// TIA Portal V16 export
// export: Created 2021-12-01T20:36:20.7617108Z, ExportSetting WithDefaults, DisplayName Totally Integrated Automation Portal, DisplayVersion V16 Update 4, DisplayName TIA Portal Version Control Interface, DisplayVersion V16 Update 2, DisplayName TIA Portal Openness, DisplayVersion V16 Update 4, DisplayName SINAMICS Startdrive Advanced, DisplayVersion V16 Update 5, DisplayName SINAMICS Startdrive G130, G150, S120, S150, SINAMICS MV, S210, DisplayVersion V16 Update 5, DisplayName SINAMICS Startdrive G110M, G120, G120C, G120D, G120P, G115D, DisplayVersion V16 Update 5, DisplayName STEP 7 Professional, DisplayVersion V16 Update 4, DisplayName STEP 7 Safety, DisplayVersion V16, DisplayName WinCC Advanced, DisplayVersion V16 Update 4
FUNCTION "ST00240_2_FC" : Void   // FC124, LAD
TITLE = ST00240_2
{ S7_Optimized_Access := 'TRUE' }
VERSION : 0.1
// stored: AutoNumber true, IsIECCheckEnabled false, SetENOAutomatically false, UDAEnableTagReadback false
   VAR_IN_OUT
      OPMODE : "OPMODE_OUT_UDT";
      HMI_EXTENSION : "HMI_EXTENSION_PANEL_UDT";
   END_VAR
   VAR_TEMP
      EmptyHS : "RT_HANDSHAKE_UDT";
   END_VAR
BEGIN

REGION Network 1: Alarm
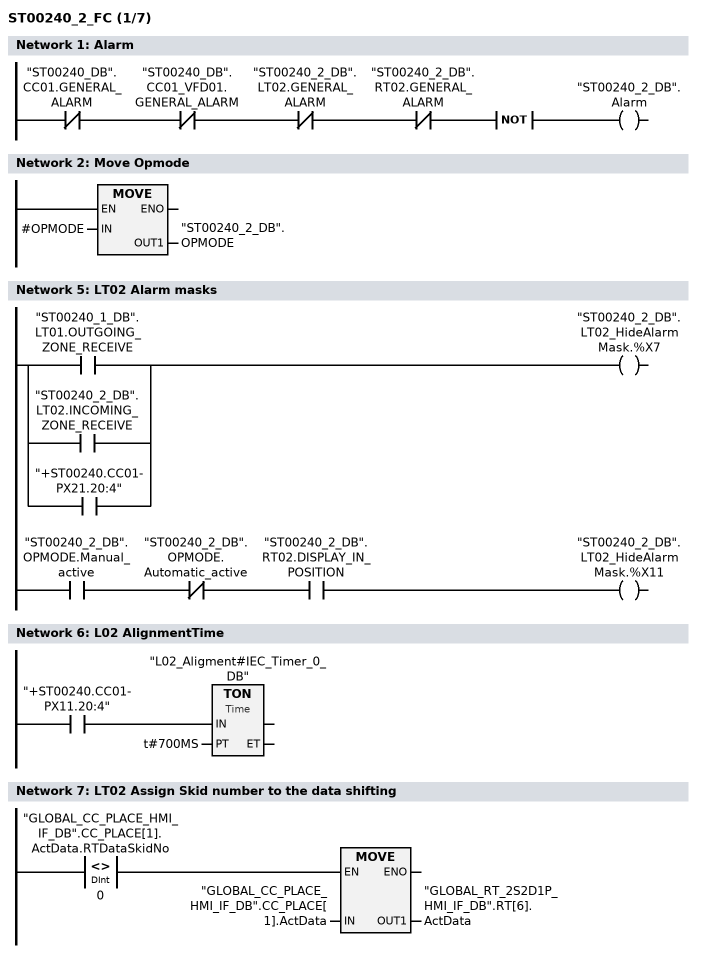
   RUNG wire#powerrail
      I_Contact( "ST00240_DB".CC01.GENERAL_ALARM )
      I_Contact( "ST00240_DB".CC01_VFD01.GENERAL_ALARM )
      I_Contact( "ST00240_2_DB".LT02.GENERAL_ALARM )
      I_Contact( "ST00240_2_DB".RT02.GENERAL_ALARM )
      Not()
      Coil( "ST00240_2_DB".Alarm )
   END_RUNG
   // the same network as SCL:
   "ST00240_2_DB".Alarm := NOT (NOT "ST00240_DB".CC01.GENERAL_ALARM AND NOT "ST00240_DB".CC01_VFD01.GENERAL_ALARM AND NOT "ST00240_2_DB".LT02.GENERAL_ALARM AND NOT "ST00240_2_DB".RT02.GENERAL_ALARM);
END_REGION

REGION Network 2: Move Opmode
   RUNG wire#powerrail
      Move(in := #OPMODE, out1 => "ST00240_2_DB".OPMODE)
   END_RUNG
   // the same network as SCL:
   "ST00240_2_DB".OPMODE := #OPMODE;
END_REGION

REGION Network 3: *******************LT02 Control*******************
END_REGION

REGION Network 4 (SCL): LT02 Parameters
   "ST00240_2_DB".LT02.PARA_SET.Para.HasMidPosition := true;
   "ST00240_2_DB".LT02.PARA_SET.Para.HasRT := TRUE;
   "ST00240_2_DB".LT02.PARA_SET.Para.PosCCStopForward := true;
   "ST00240_2_DB".LT02.PARA_SET.Para.PosCCStopReverse := false;
   "ST00240_2_DB".LT02.PARA_SET.Para.PosRaiseForward_1 := true;
   "ST00240_2_DB".LT02.PARA_SET.Para.PosRaiseForward_2 := true;
   "ST00240_2_DB".LT02.PARA_SET.Para.PosRaiseReverse_1 := true;
   "ST00240_2_DB".LT02.PARA_SET.Para.PosRaiseReverse_2 := false;
   "ST00240_2_DB".LT02.PARA_SET.Para.PosSlowForward := true;
   "ST00240_2_DB".LT02.PARA_SET.Para.PosSlowReverse := false;
   "ST00240_2_DB".LT02.PARA_SET.Set.RuntimeLower := t#10s;
   "ST00240_2_DB".LT02.PARA_SET.Set.RuntimeLift := t#11s;
   "ST00240_2_DB".LT02.PARA_SET.Set.AlignmentTime := t#0ms;
END_REGION

REGION Network 5: LT02 Alarm masks
   RUNG wire#powerrail
      Contact( "ST00240_1_DB".LT01.OUTGOING_ZONE_RECEIVE )
      wire#w1
      Coil( "ST00240_2_DB".LT02_HideAlarmMask.%X7 )
   END_RUNG
   RUNG wire#powerrail
      Contact( "ST00240_2_DB".LT02.INCOMING_ZONE_RECEIVE )
   END_RUNG wire#w1
   RUNG wire#powerrail
      Contact( "+ST00240.CC01-PX21.20:4" )
   END_RUNG wire#w1
   RUNG wire#powerrail
      Contact( "ST00240_2_DB".OPMODE.Manual_active )
      I_Contact( "ST00240_2_DB".OPMODE.Automatic_active )
      Contact( "ST00240_2_DB".RT02.DISPLAY_IN_POSITION )
      Coil( "ST00240_2_DB".LT02_HideAlarmMask.%X11 )
   END_RUNG
   // the same network as SCL:
   "ST00240_2_DB".LT02_HideAlarmMask.%X7 := "ST00240_1_DB".LT01.OUTGOING_ZONE_RECEIVE OR "ST00240_2_DB".LT02.INCOMING_ZONE_RECEIVE OR "+ST00240.CC01-PX21.20:4";
   "ST00240_2_DB".LT02_HideAlarmMask.%X11 := "ST00240_2_DB".OPMODE.Manual_active AND NOT "ST00240_2_DB".OPMODE.Automatic_active AND "ST00240_2_DB".RT02.DISPLAY_IN_POSITION;
END_REGION

REGION Network 6: L02 AlignmentTime
   RUNG wire#powerrail
      Contact( "+ST00240.CC01-PX11.20:4" )
      { S7_Templates := "time_type := Time" } "L02_Aligment#IEC_Timer_0_DB".TON(pt := t#700MS, et =>)
   END_RUNG
   // the same network as SCL:
   "L02_Aligment#IEC_Timer_0_DB".TON(IN := "+ST00240.CC01-PX11.20:4", PT := t#700MS);
END_REGION

REGION Network 7: LT02 Assign Skid number to the data shifting
   RUNG wire#powerrail
      { S7_Templates := "SrcType := DInt" } NE_Contact(in1 := "GLOBAL_CC_PLACE_HMI_IF_DB".CC_PLACE[1].ActData.RTDataSkidNo, in2 := 0)
      Move(in := "GLOBAL_CC_PLACE_HMI_IF_DB".CC_PLACE[1].ActData, out1 => "GLOBAL_RT_2S2D1P_HMI_IF_DB".RT[6].ActData)
   END_RUNG
   // the same network as SCL:
   IF "GLOBAL_CC_PLACE_HMI_IF_DB".CC_PLACE[1].ActData.RTDataSkidNo <> 0 THEN
       "GLOBAL_RT_2S2D1P_HMI_IF_DB".RT[6].ActData := "GLOBAL_CC_PLACE_HMI_IF_DB".CC_PLACE[1].ActData;
   END_IF;
END_REGION

REGION Network 8: LT02 CC Place FB
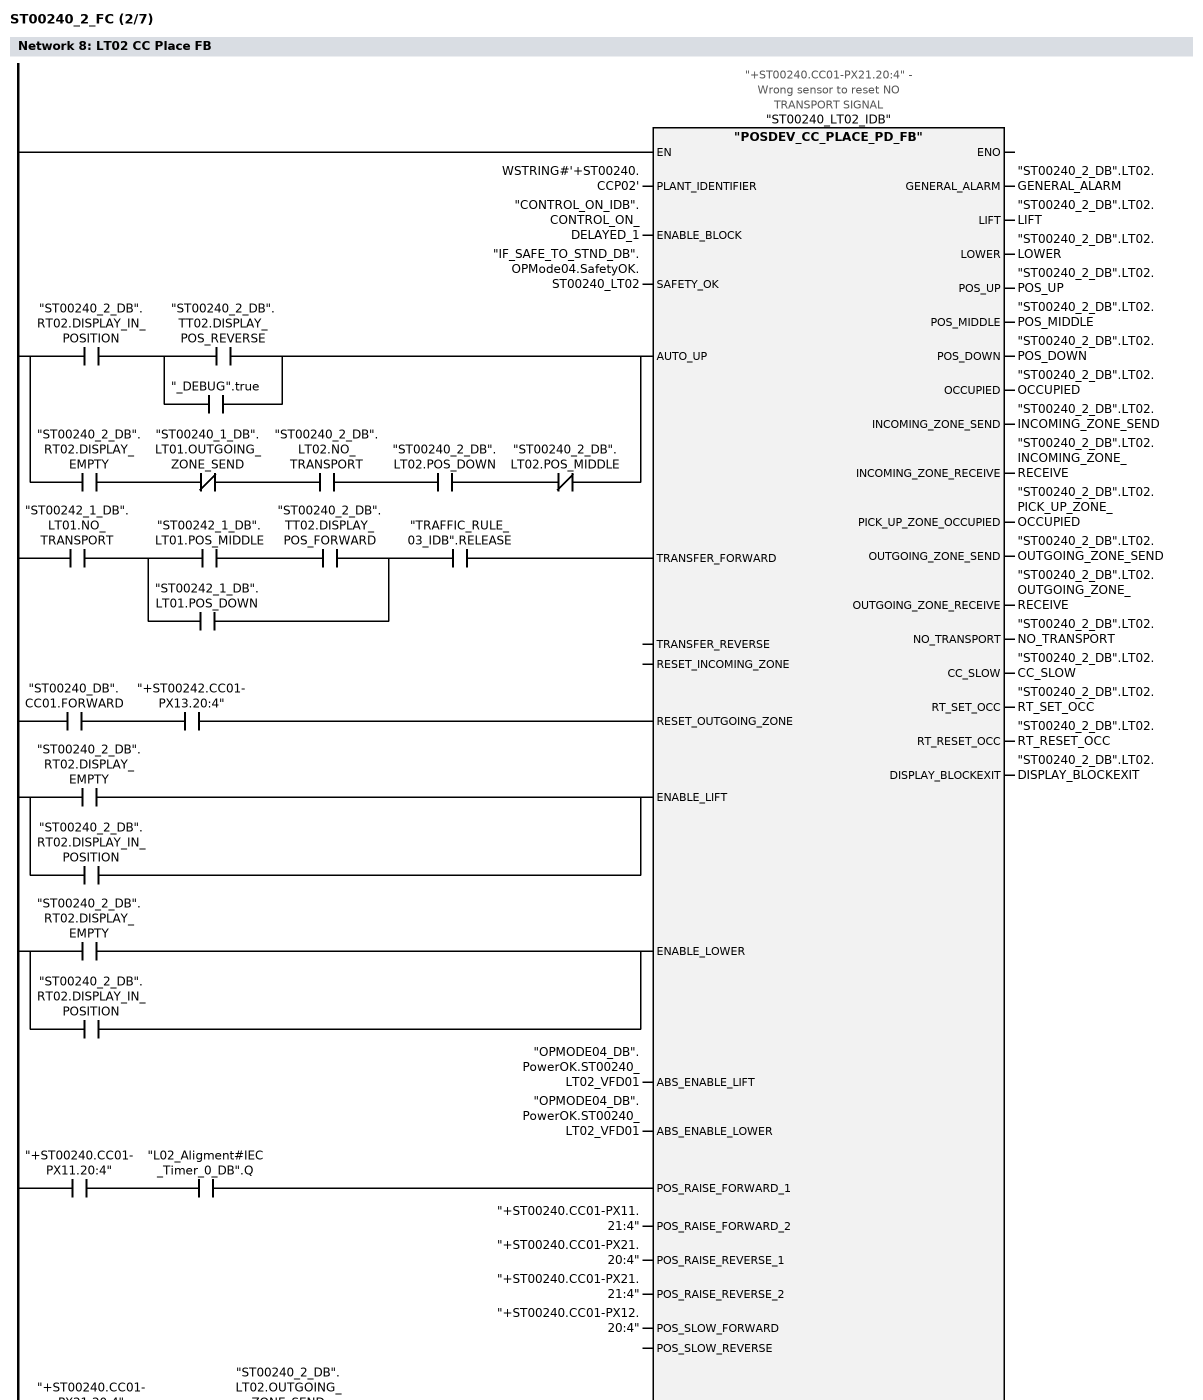
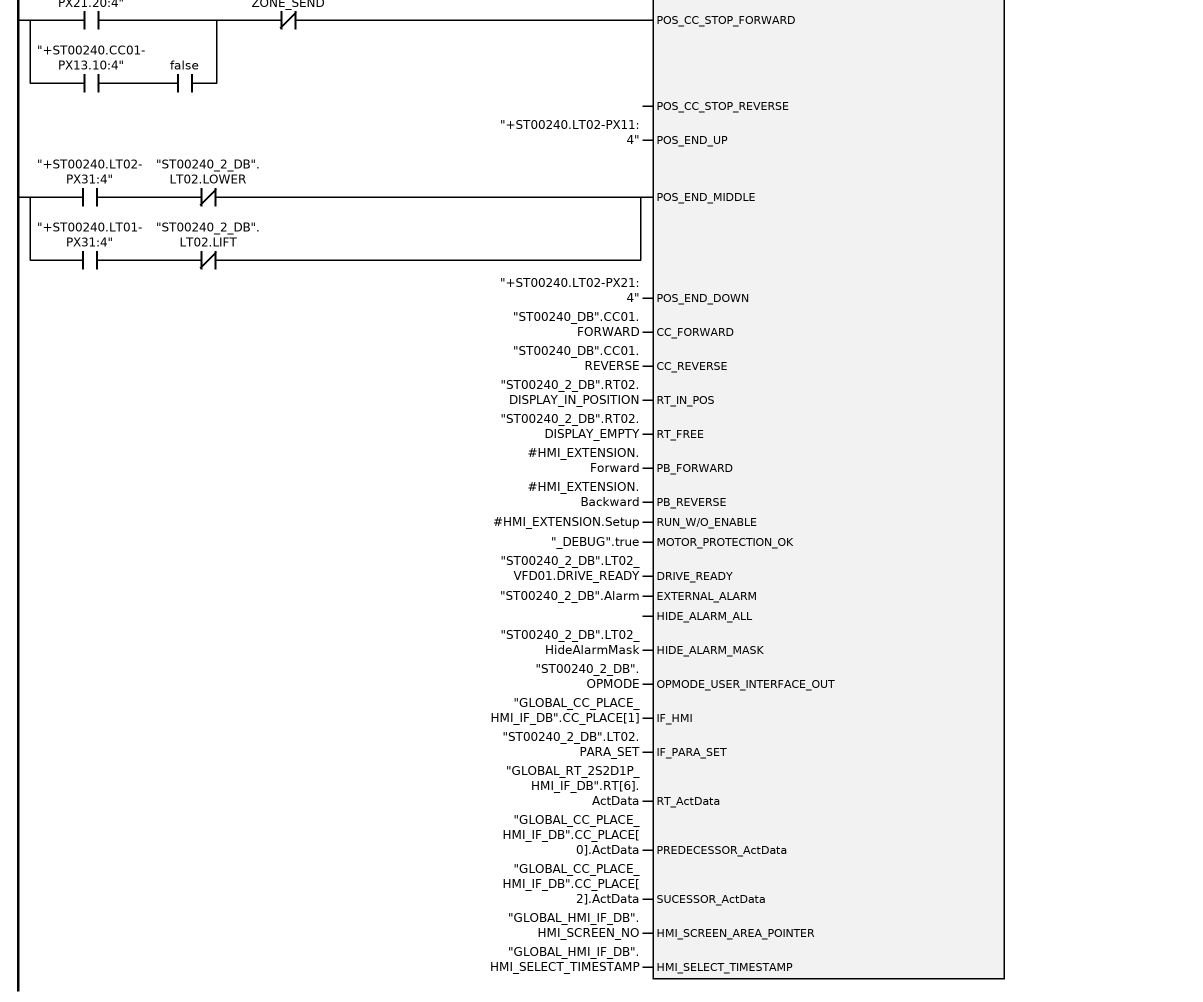
   RUNG wire#powerrail
      "ST00240_LT02_IDB"(AUTO_UP := wire#w2, TRANSFER_FORWARD := wire#w5, RESET_OUTGOING_ZONE := wire#w6, ENABLE_LIFT := wire#w7, ENABLE_LOWER := wire#w8, POS_RAISE_FORWARD_1 := wire#w9, POS_CC_STOP_FORWARD := wire#w11, POS_END_MIDDLE := wire#w12, PLANT_IDENTIFIER := WSTRING#'+ST00240.CCP02', ENABLE_BLOCK := "CONTROL_ON_IDB".CONTROL_ON_DELAYED_1, SAFETY_OK := "IF_SAFE_TO_STND_DB".OPMode04.SafetyOK.ST00240_LT02, TRANSFER_REVERSE :=, RESET_INCOMING_ZONE :=, ABS_ENABLE_LIFT := "OPMODE04_DB".PowerOK.ST00240_LT02_VFD01, ABS_ENABLE_LOWER := "OPMODE04_DB".PowerOK.ST00240_LT02_VFD01, POS_RAISE_FORWARD_2 := "+ST00240.CC01-PX11.21:4", POS_RAISE_REVERSE_1 := "+ST00240.CC01-PX21.20:4", POS_RAISE_REVERSE_2 := "+ST00240.CC01-PX21.21:4", POS_SLOW_FORWARD := "+ST00240.CC01-PX12.20:4", POS_SLOW_REVERSE :=, POS_CC_STOP_REVERSE :=, POS_END_UP := "+ST00240.LT02-PX11:4", POS_END_DOWN := "+ST00240.LT02-PX21:4", CC_FORWARD := "ST00240_DB".CC01.FORWARD, CC_REVERSE := "ST00240_DB".CC01.REVERSE, RT_IN_POS := "ST00240_2_DB".RT02.DISPLAY_IN_POSITION, RT_FREE := "ST00240_2_DB".RT02.DISPLAY_EMPTY, PB_FORWARD := #HMI_EXTENSION.Forward, PB_REVERSE := #HMI_EXTENSION.Backward, "RUN_W/O_ENABLE" := #HMI_EXTENSION.Setup, MOTOR_PROTECTION_OK := "_DEBUG".true, DRIVE_READY := "ST00240_2_DB".LT02_VFD01.DRIVE_READY, EXTERNAL_ALARM := "ST00240_2_DB".Alarm, HIDE_ALARM_ALL :=, HIDE_ALARM_MASK := "ST00240_2_DB".LT02_HideAlarmMask, OPMODE_USER_INTERFACE_OUT := "ST00240_2_DB".OPMODE, IF_HMI := "GLOBAL_CC_PLACE_HMI_IF_DB".CC_PLACE[1], IF_PARA_SET := "ST00240_2_DB".LT02.PARA_SET, RT_ActData := "GLOBAL_RT_2S2D1P_HMI_IF_DB".RT[6].ActData, PREDECESSOR_ActData := "GLOBAL_CC_PLACE_HMI_IF_DB".CC_PLACE[0].ActData, SUCESSOR_ActData := "GLOBAL_CC_PLACE_HMI_IF_DB".CC_PLACE[2].ActData, HMI_SCREEN_AREA_POINTER := "GLOBAL_HMI_IF_DB".HMI_SCREEN_NO, HMI_SELECT_TIMESTAMP := "GLOBAL_HMI_IF_DB".HMI_SELECT_TIMESTAMP, GENERAL_ALARM => "ST00240_2_DB".LT02.GENERAL_ALARM, LIFT => "ST00240_2_DB".LT02.LIFT, LOWER => "ST00240_2_DB".LT02.LOWER, POS_UP => "ST00240_2_DB".LT02.POS_UP, POS_MIDDLE => "ST00240_2_DB".LT02.POS_MIDDLE, POS_DOWN => "ST00240_2_DB".LT02.POS_DOWN, OCCUPIED => "ST00240_2_DB".LT02.OCCUPIED, INCOMING_ZONE_SEND => "ST00240_2_DB".LT02.INCOMING_ZONE_SEND, INCOMING_ZONE_RECEIVE => "ST00240_2_DB".LT02.INCOMING_ZONE_RECEIVE, PICK_UP_ZONE_OCCUPIED => "ST00240_2_DB".LT02.PICK_UP_ZONE_OCCUPIED, OUTGOING_ZONE_SEND => "ST00240_2_DB".LT02.OUTGOING_ZONE_SEND, OUTGOING_ZONE_RECEIVE => "ST00240_2_DB".LT02.OUTGOING_ZONE_RECEIVE, NO_TRANSPORT => "ST00240_2_DB".LT02.NO_TRANSPORT, CC_SLOW => "ST00240_2_DB".LT02.CC_SLOW, RT_SET_OCC => "ST00240_2_DB".LT02.RT_SET_OCC, RT_RESET_OCC => "ST00240_2_DB".LT02.RT_RESET_OCC, DISPLAY_BLOCKEXIT => "ST00240_2_DB".LT02.DISPLAY_BLOCKEXIT)   // "+ST00240.CC01-PX21.20:4" - Wrong sensor to reset NO TRANSPORT SIGNAL
   END_RUNG
   RUNG wire#powerrail
      Contact( "ST00240_2_DB".RT02.DISPLAY_IN_POSITION )
      wire#w1
      Contact( "ST00240_2_DB".TT02.DISPLAY_POS_REVERSE )
   END_RUNG wire#w2
   RUNG wire#w1
      Contact( "_DEBUG".true )
   END_RUNG wire#w2
   RUNG wire#powerrail
      Contact( "ST00240_2_DB".RT02.DISPLAY_EMPTY )
      I_Contact( "ST00240_1_DB".LT01.OUTGOING_ZONE_SEND )
      Contact( "ST00240_2_DB".LT02.NO_TRANSPORT )
      Contact( "ST00240_2_DB".LT02.POS_DOWN )
      I_Contact( "ST00240_2_DB".LT02.POS_MIDDLE )
   END_RUNG wire#w2
   RUNG wire#powerrail
      Contact( "ST00242_1_DB".LT01.NO_TRANSPORT )
      wire#w3
      Contact( "ST00242_1_DB".LT01.POS_MIDDLE )
      Contact( "ST00240_2_DB".TT02.DISPLAY_POS_FORWARD )
      wire#w4
      Contact( "TRAFFIC_RULE_03_IDB".RELEASE )
   END_RUNG wire#w5
   RUNG wire#w3
      Contact( "ST00242_1_DB".LT01.POS_DOWN )
   END_RUNG wire#w4
   RUNG wire#powerrail
      Contact( "ST00240_DB".CC01.FORWARD )
      Contact( "+ST00242.CC01-PX13.20:4" )
   END_RUNG wire#w6
   RUNG wire#powerrail
      Contact( "ST00240_2_DB".RT02.DISPLAY_EMPTY )
   END_RUNG wire#w7
   RUNG wire#powerrail
      Contact( "ST00240_2_DB".RT02.DISPLAY_IN_POSITION )
   END_RUNG wire#w7
   RUNG wire#powerrail
      Contact( "ST00240_2_DB".RT02.DISPLAY_EMPTY )
   END_RUNG wire#w8
   RUNG wire#powerrail
      Contact( "ST00240_2_DB".RT02.DISPLAY_IN_POSITION )
   END_RUNG wire#w8
   RUNG wire#powerrail
      Contact( "+ST00240.CC01-PX11.20:4" )
      Contact( "L02_Aligment#IEC_Timer_0_DB".Q )
   END_RUNG wire#w9
   RUNG wire#powerrail
      Contact( "+ST00240.CC01-PX21.20:4" )
      wire#w10
      I_Contact( "ST00240_2_DB".LT02.OUTGOING_ZONE_SEND )
   END_RUNG wire#w11
   RUNG wire#powerrail
      Contact( "+ST00240.CC01-PX13.10:4" )
      Contact( false )
   END_RUNG wire#w10
   RUNG wire#powerrail
      Contact( "+ST00240.LT02-PX31:4" )
      I_Contact( "ST00240_2_DB".LT02.LOWER )
   END_RUNG wire#w12
   RUNG wire#powerrail
      Contact( "+ST00240.LT01-PX31:4" )
      I_Contact( "ST00240_2_DB".LT02.LIFT )
   END_RUNG wire#w12
   // the same network as SCL:
   "ST00240_LT02_IDB"(PLANT_IDENTIFIER := WSTRING#'+ST00240.CCP02',   // "POSDEV_CC_PLACE_PD_FB": "+ST00240.CC01-PX21.20:4" - Wrong sensor to reset NO TRANSPORT SIGNAL
                      ENABLE_BLOCK := "CONTROL_ON_IDB".CONTROL_ON_DELAYED_1,
                      SAFETY_OK := "IF_SAFE_TO_STND_DB".OPMode04.SafetyOK.ST00240_LT02,
                      AUTO_UP := ("ST00240_2_DB".RT02.DISPLAY_IN_POSITION AND ("ST00240_2_DB".TT02.DISPLAY_POS_REVERSE OR "_DEBUG".true)) OR ("ST00240_2_DB".RT02.DISPLAY_EMPTY AND NOT "ST00240_1_DB".LT01.OUTGOING_ZONE_SEND AND "ST00240_2_DB".LT02.NO_TRANSPORT AND "ST00240_2_DB".LT02.POS_DOWN AND NOT "ST00240_2_DB".LT02.POS_MIDDLE),
                      TRANSFER_FORWARD := "ST00242_1_DB".LT01.NO_TRANSPORT AND (("ST00242_1_DB".LT01.POS_MIDDLE AND "ST00240_2_DB".TT02.DISPLAY_POS_FORWARD) OR "ST00242_1_DB".LT01.POS_DOWN) AND "TRAFFIC_RULE_03_IDB".RELEASE,
                      RESET_OUTGOING_ZONE := "ST00240_DB".CC01.FORWARD AND "+ST00242.CC01-PX13.20:4",
                      ENABLE_LIFT := "ST00240_2_DB".RT02.DISPLAY_EMPTY OR "ST00240_2_DB".RT02.DISPLAY_IN_POSITION,
                      ENABLE_LOWER := "ST00240_2_DB".RT02.DISPLAY_EMPTY OR "ST00240_2_DB".RT02.DISPLAY_IN_POSITION,
                      ABS_ENABLE_LIFT := "OPMODE04_DB".PowerOK.ST00240_LT02_VFD01,
                      ABS_ENABLE_LOWER := "OPMODE04_DB".PowerOK.ST00240_LT02_VFD01,
                      POS_RAISE_FORWARD_1 := "+ST00240.CC01-PX11.20:4" AND "L02_Aligment#IEC_Timer_0_DB".Q,
                      POS_RAISE_FORWARD_2 := "+ST00240.CC01-PX11.21:4",
                      POS_RAISE_REVERSE_1 := "+ST00240.CC01-PX21.20:4",
                      POS_RAISE_REVERSE_2 := "+ST00240.CC01-PX21.21:4",
                      POS_SLOW_FORWARD := "+ST00240.CC01-PX12.20:4",
                      POS_CC_STOP_FORWARD := ("+ST00240.CC01-PX21.20:4" OR ("+ST00240.CC01-PX13.10:4" AND false)) AND NOT "ST00240_2_DB".LT02.OUTGOING_ZONE_SEND,
                      POS_END_UP := "+ST00240.LT02-PX11:4",
                      POS_END_MIDDLE := ("+ST00240.LT02-PX31:4" AND NOT "ST00240_2_DB".LT02.LOWER) OR ("+ST00240.LT01-PX31:4" AND NOT "ST00240_2_DB".LT02.LIFT),
                      POS_END_DOWN := "+ST00240.LT02-PX21:4",
                      CC_FORWARD := "ST00240_DB".CC01.FORWARD,
                      CC_REVERSE := "ST00240_DB".CC01.REVERSE,
                      RT_IN_POS := "ST00240_2_DB".RT02.DISPLAY_IN_POSITION,
                      RT_FREE := "ST00240_2_DB".RT02.DISPLAY_EMPTY,
                      PB_FORWARD := #HMI_EXTENSION.Forward,
                      PB_REVERSE := #HMI_EXTENSION.Backward,
                      "RUN_W/O_ENABLE" := #HMI_EXTENSION.Setup,
                      MOTOR_PROTECTION_OK := "_DEBUG".true,
                      DRIVE_READY := "ST00240_2_DB".LT02_VFD01.DRIVE_READY,
                      EXTERNAL_ALARM := "ST00240_2_DB".Alarm,
                      HIDE_ALARM_MASK := "ST00240_2_DB".LT02_HideAlarmMask,
                      OPMODE_USER_INTERFACE_OUT := "ST00240_2_DB".OPMODE,
                      IF_HMI := "GLOBAL_CC_PLACE_HMI_IF_DB".CC_PLACE[1],
                      IF_PARA_SET := "ST00240_2_DB".LT02.PARA_SET,
                      RT_ActData := "GLOBAL_RT_2S2D1P_HMI_IF_DB".RT[6].ActData,
                      PREDECESSOR_ActData := "GLOBAL_CC_PLACE_HMI_IF_DB".CC_PLACE[0].ActData,
                      SUCESSOR_ActData := "GLOBAL_CC_PLACE_HMI_IF_DB".CC_PLACE[2].ActData,
                      HMI_SCREEN_AREA_POINTER := "GLOBAL_HMI_IF_DB".HMI_SCREEN_NO,
                      HMI_SELECT_TIMESTAMP := "GLOBAL_HMI_IF_DB".HMI_SELECT_TIMESTAMP,
                      GENERAL_ALARM => "ST00240_2_DB".LT02.GENERAL_ALARM,
                      LIFT => "ST00240_2_DB".LT02.LIFT,
                      LOWER => "ST00240_2_DB".LT02.LOWER,
                      POS_UP => "ST00240_2_DB".LT02.POS_UP,
                      POS_MIDDLE => "ST00240_2_DB".LT02.POS_MIDDLE,
                      POS_DOWN => "ST00240_2_DB".LT02.POS_DOWN,
                      OCCUPIED => "ST00240_2_DB".LT02.OCCUPIED,
                      INCOMING_ZONE_SEND => "ST00240_2_DB".LT02.INCOMING_ZONE_SEND,
                      INCOMING_ZONE_RECEIVE => "ST00240_2_DB".LT02.INCOMING_ZONE_RECEIVE,
                      PICK_UP_ZONE_OCCUPIED => "ST00240_2_DB".LT02.PICK_UP_ZONE_OCCUPIED,
                      OUTGOING_ZONE_SEND => "ST00240_2_DB".LT02.OUTGOING_ZONE_SEND,
                      OUTGOING_ZONE_RECEIVE => "ST00240_2_DB".LT02.OUTGOING_ZONE_RECEIVE,
                      NO_TRANSPORT => "ST00240_2_DB".LT02.NO_TRANSPORT,
                      CC_SLOW => "ST00240_2_DB".LT02.CC_SLOW,
                      RT_SET_OCC => "ST00240_2_DB".LT02.RT_SET_OCC,
                      RT_RESET_OCC => "ST00240_2_DB".LT02.RT_RESET_OCC,
                      DISPLAY_BLOCKEXIT => "ST00240_2_DB".LT02.DISPLAY_BLOCKEXIT);
END_REGION

REGION Network 9: LT02 Speed
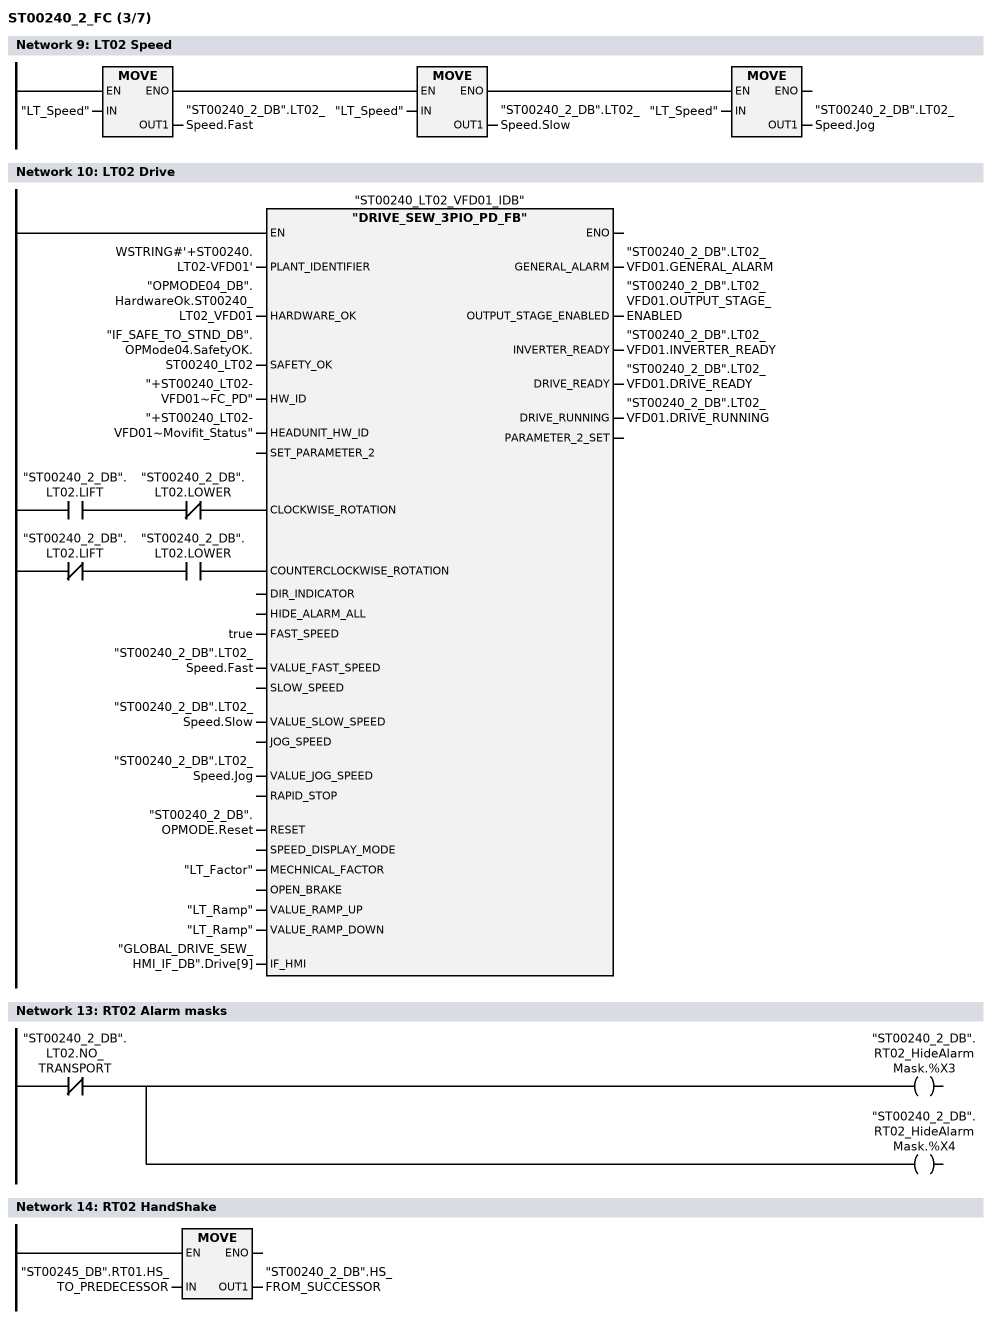
   RUNG wire#powerrail
      Move(in := "LT_Speed", out1 => "ST00240_2_DB".LT02_Speed.Fast)
      Move(in := "LT_Speed", out1 => "ST00240_2_DB".LT02_Speed.Slow)
      Move(in := "LT_Speed", out1 => "ST00240_2_DB".LT02_Speed.Jog)
   END_RUNG
   // the same network as SCL:
   "ST00240_2_DB".LT02_Speed.Fast := "LT_Speed";
   "ST00240_2_DB".LT02_Speed.Slow := "LT_Speed";
   "ST00240_2_DB".LT02_Speed.Jog := "LT_Speed";
END_REGION

REGION Network 10: LT02 Drive
   RUNG wire#powerrail
      "ST00240_LT02_VFD01_IDB"(CLOCKWISE_ROTATION := wire#w1, COUNTERCLOCKWISE_ROTATION := wire#w2, PLANT_IDENTIFIER := WSTRING#'+ST00240.LT02-VFD01', HARDWARE_OK := "OPMODE04_DB".HardwareOk.ST00240_LT02_VFD01, SAFETY_OK := "IF_SAFE_TO_STND_DB".OPMode04.SafetyOK.ST00240_LT02, HW_ID := "+ST00240_LT02-VFD01~FC_PD", HEADUNIT_HW_ID := "+ST00240_LT02-VFD01~Movifit_Status", SET_PARAMETER_2 :=, DIR_INDICATOR :=, HIDE_ALARM_ALL :=, FAST_SPEED := true, VALUE_FAST_SPEED := "ST00240_2_DB".LT02_Speed.Fast, SLOW_SPEED :=, VALUE_SLOW_SPEED := "ST00240_2_DB".LT02_Speed.Slow, JOG_SPEED :=, VALUE_JOG_SPEED := "ST00240_2_DB".LT02_Speed.Jog, RAPID_STOP :=, RESET := "ST00240_2_DB".OPMODE.Reset, SPEED_DISPLAY_MODE :=, MECHNICAL_FACTOR := "LT_Factor", OPEN_BRAKE :=, VALUE_RAMP_UP := "LT_Ramp", VALUE_RAMP_DOWN := "LT_Ramp", IF_HMI := "GLOBAL_DRIVE_SEW_HMI_IF_DB".Drive[9], GENERAL_ALARM => "ST00240_2_DB".LT02_VFD01.GENERAL_ALARM, OUTPUT_STAGE_ENABLED => "ST00240_2_DB".LT02_VFD01.OUTPUT_STAGE_ENABLED, INVERTER_READY => "ST00240_2_DB".LT02_VFD01.INVERTER_READY, DRIVE_READY => "ST00240_2_DB".LT02_VFD01.DRIVE_READY, DRIVE_RUNNING => "ST00240_2_DB".LT02_VFD01.DRIVE_RUNNING, PARAMETER_2_SET =>)
   END_RUNG
   RUNG wire#powerrail
      Contact( "ST00240_2_DB".LT02.LIFT )
      I_Contact( "ST00240_2_DB".LT02.LOWER )
   END_RUNG wire#w1
   RUNG wire#powerrail
      I_Contact( "ST00240_2_DB".LT02.LIFT )
      Contact( "ST00240_2_DB".LT02.LOWER )
   END_RUNG wire#w2
   // the same network as SCL:
   "ST00240_LT02_VFD01_IDB"(PLANT_IDENTIFIER := WSTRING#'+ST00240.LT02-VFD01',   // "DRIVE_SEW_3PIO_PD_FB"
                           HARDWARE_OK := "OPMODE04_DB".HardwareOk.ST00240_LT02_VFD01,
                           SAFETY_OK := "IF_SAFE_TO_STND_DB".OPMode04.SafetyOK.ST00240_LT02,
                           HW_ID := "+ST00240_LT02-VFD01~FC_PD",
                           HEADUNIT_HW_ID := "+ST00240_LT02-VFD01~Movifit_Status",
                           CLOCKWISE_ROTATION := "ST00240_2_DB".LT02.LIFT AND NOT "ST00240_2_DB".LT02.LOWER,
                           COUNTERCLOCKWISE_ROTATION := NOT "ST00240_2_DB".LT02.LIFT AND "ST00240_2_DB".LT02.LOWER,
                           FAST_SPEED := true,
                           VALUE_FAST_SPEED := "ST00240_2_DB".LT02_Speed.Fast,
                           VALUE_SLOW_SPEED := "ST00240_2_DB".LT02_Speed.Slow,
                           VALUE_JOG_SPEED := "ST00240_2_DB".LT02_Speed.Jog,
                           RESET := "ST00240_2_DB".OPMODE.Reset,
                           MECHNICAL_FACTOR := "LT_Factor",
                           VALUE_RAMP_UP := "LT_Ramp",
                           VALUE_RAMP_DOWN := "LT_Ramp",
                           IF_HMI := "GLOBAL_DRIVE_SEW_HMI_IF_DB".Drive[9],
                           GENERAL_ALARM => "ST00240_2_DB".LT02_VFD01.GENERAL_ALARM,
                           OUTPUT_STAGE_ENABLED => "ST00240_2_DB".LT02_VFD01.OUTPUT_STAGE_ENABLED,
                           INVERTER_READY => "ST00240_2_DB".LT02_VFD01.INVERTER_READY,
                           DRIVE_READY => "ST00240_2_DB".LT02_VFD01.DRIVE_READY,
                           DRIVE_RUNNING => "ST00240_2_DB".LT02_VFD01.DRIVE_RUNNING);
END_REGION

REGION Network 11: *******************RT02 Control*******************
END_REGION

REGION Network 12 (SCL): RT02 Parameters
   "ST00240_2_DB".RT02.PARA_SET.Para.PosEndForward1 := true;
   "ST00240_2_DB".RT02.PARA_SET.Para.PosEndReverse := true;
   "ST00240_2_DB".RT02.PARA_SET.Para.PosSlowForward := false;

   "ST00240_2_DB".RT02.PARA_SET.Set.RunTimeForward := 450;
   "ST00240_2_DB".RT02.PARA_SET.Set.RunTimeReverse := 450;
END_REGION

REGION Network 13: RT02 Alarm masks
   RUNG wire#powerrail
      I_Contact( "ST00240_2_DB".LT02.NO_TRANSPORT )
      wire#w1
      Coil( "ST00240_2_DB".RT02_HideAlarmMask.%X3 )
   END_RUNG
   RUNG wire#w1
      Coil( "ST00240_2_DB".RT02_HideAlarmMask.%X4 )
   END_RUNG
   // the same network as SCL:
   "ST00240_2_DB".RT02_HideAlarmMask.%X3 := NOT "ST00240_2_DB".LT02.NO_TRANSPORT;
   "ST00240_2_DB".RT02_HideAlarmMask.%X4 := NOT "ST00240_2_DB".LT02.NO_TRANSPORT;
END_REGION

REGION Network 14: RT02 HandShake
   RUNG wire#powerrail
      Move(in := "ST00245_DB".RT01.HS_TO_PREDECESSOR, out1 => "ST00240_2_DB".HS_FROM_SUCCESSOR)
   END_RUNG
   // the same network as SCL:
   "ST00240_2_DB".HS_FROM_SUCCESSOR := "ST00245_DB".RT01.HS_TO_PREDECESSOR;
END_REGION

REGION Network 15: RT02 FB Control
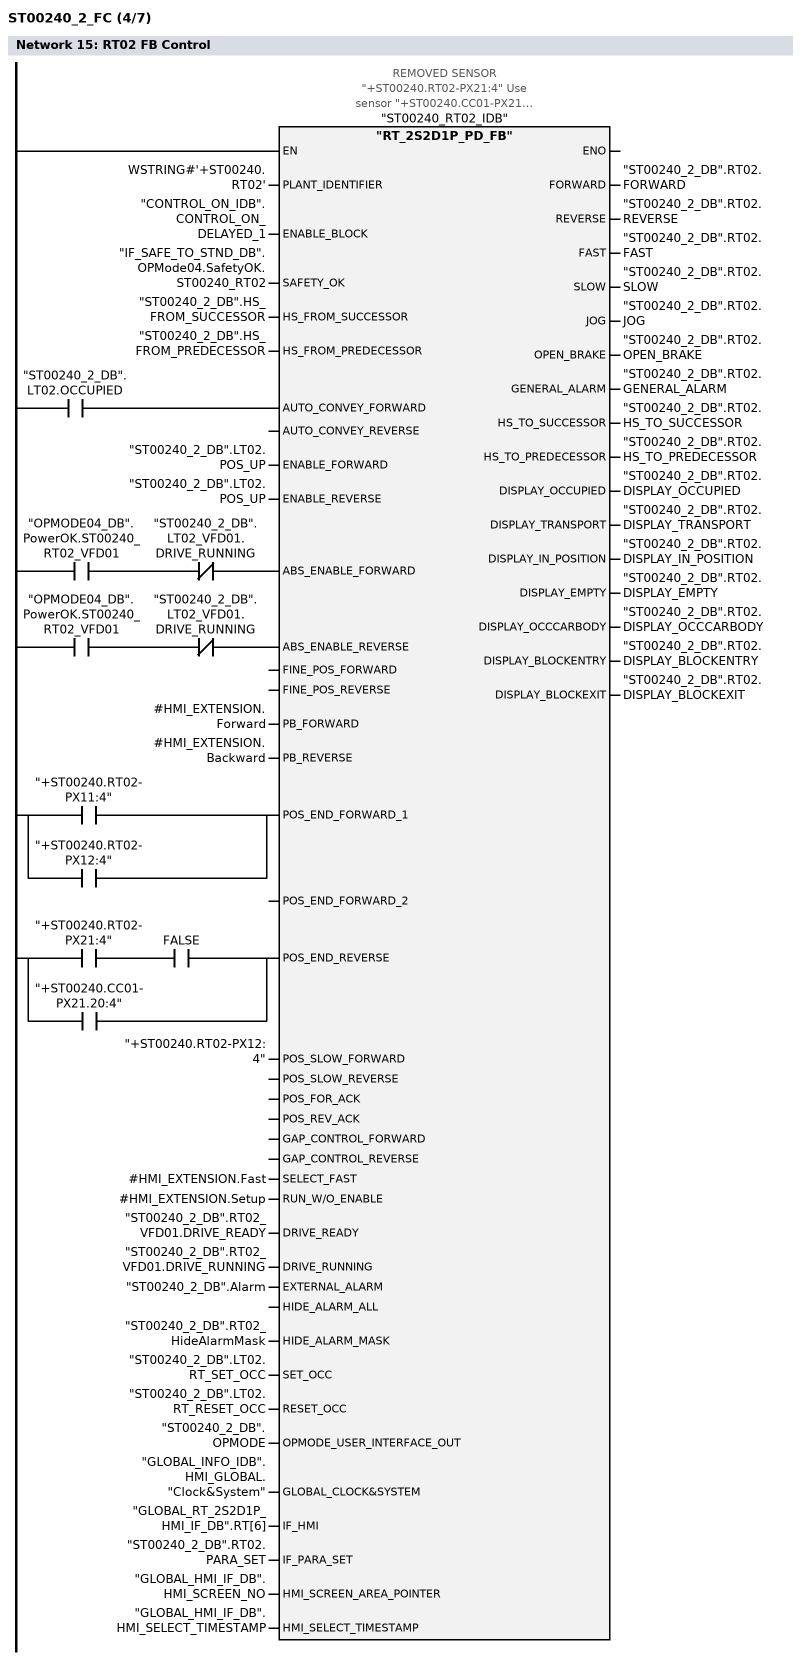
   RUNG wire#powerrail
      "ST00240_RT02_IDB"(AUTO_CONVEY_FORWARD := wire#w1, ABS_ENABLE_FORWARD := wire#w2, ABS_ENABLE_REVERSE := wire#w3, POS_END_FORWARD_1 := wire#w4, POS_END_REVERSE := wire#w5, PLANT_IDENTIFIER := WSTRING#'+ST00240.RT02', ENABLE_BLOCK := "CONTROL_ON_IDB".CONTROL_ON_DELAYED_1, SAFETY_OK := "IF_SAFE_TO_STND_DB".OPMode04.SafetyOK.ST00240_RT02, HS_FROM_SUCCESSOR := "ST00240_2_DB".HS_FROM_SUCCESSOR, HS_FROM_PREDECESSOR := "ST00240_2_DB".HS_FROM_PREDECESSOR, AUTO_CONVEY_REVERSE :=, ENABLE_FORWARD := "ST00240_2_DB".LT02.POS_UP, ENABLE_REVERSE := "ST00240_2_DB".LT02.POS_UP, FINE_POS_FORWARD :=, FINE_POS_REVERSE :=, PB_FORWARD := #HMI_EXTENSION.Forward, PB_REVERSE := #HMI_EXTENSION.Backward, POS_END_FORWARD_2 :=, POS_SLOW_FORWARD := "+ST00240.RT02-PX12:4", POS_SLOW_REVERSE :=, POS_FOR_ACK :=, POS_REV_ACK :=, GAP_CONTROL_FORWARD :=, GAP_CONTROL_REVERSE :=, SELECT_FAST := #HMI_EXTENSION.Fast, "RUN_W/O_ENABLE" := #HMI_EXTENSION.Setup, DRIVE_READY := "ST00240_2_DB".RT02_VFD01.DRIVE_READY, DRIVE_RUNNING := "ST00240_2_DB".RT02_VFD01.DRIVE_RUNNING, EXTERNAL_ALARM := "ST00240_2_DB".Alarm, HIDE_ALARM_ALL :=, HIDE_ALARM_MASK := "ST00240_2_DB".RT02_HideAlarmMask, SET_OCC := "ST00240_2_DB".LT02.RT_SET_OCC, RESET_OCC := "ST00240_2_DB".LT02.RT_RESET_OCC, OPMODE_USER_INTERFACE_OUT := "ST00240_2_DB".OPMODE, "GLOBAL_CLOCK&SYSTEM" := "GLOBAL_INFO_IDB".HMI_GLOBAL."Clock&System", IF_HMI := "GLOBAL_RT_2S2D1P_HMI_IF_DB".RT[6], IF_PARA_SET := "ST00240_2_DB".RT02.PARA_SET, HMI_SCREEN_AREA_POINTER := "GLOBAL_HMI_IF_DB".HMI_SCREEN_NO, HMI_SELECT_TIMESTAMP := "GLOBAL_HMI_IF_DB".HMI_SELECT_TIMESTAMP, FORWARD => "ST00240_2_DB".RT02.FORWARD, REVERSE => "ST00240_2_DB".RT02.REVERSE, FAST => "ST00240_2_DB".RT02.FAST, SLOW => "ST00240_2_DB".RT02.SLOW, JOG => "ST00240_2_DB".RT02.JOG, OPEN_BRAKE => "ST00240_2_DB".RT02.OPEN_BRAKE, GENERAL_ALARM => "ST00240_2_DB".RT02.GENERAL_ALARM, HS_TO_SUCCESSOR => "ST00240_2_DB".RT02.HS_TO_SUCCESSOR, HS_TO_PREDECESSOR => "ST00240_2_DB".RT02.HS_TO_PREDECESSOR, DISPLAY_OCCUPIED => "ST00240_2_DB".RT02.DISPLAY_OCCUPIED, DISPLAY_TRANSPORT => "ST00240_2_DB".RT02.DISPLAY_TRANSPORT, DISPLAY_IN_POSITION => "ST00240_2_DB".RT02.DISPLAY_IN_POSITION, DISPLAY_EMPTY => "ST00240_2_DB".RT02.DISPLAY_EMPTY, DISPLAY_OCCCARBODY => "ST00240_2_DB".RT02.DISPLAY_OCCCARBODY, DISPLAY_BLOCKENTRY => "ST00240_2_DB".RT02.DISPLAY_BLOCKENTRY, DISPLAY_BLOCKEXIT => "ST00240_2_DB".RT02.DISPLAY_BLOCKEXIT)   // REMOVED SENSOR "+ST00240.RT02-PX21:4" Use sensor "+ST00240.CC01-PX21.20:4" (Same sensor for CC POS 2)
   END_RUNG
   RUNG wire#powerrail
      Contact( "ST00240_2_DB".LT02.OCCUPIED )
   END_RUNG wire#w1
   RUNG wire#powerrail
      Contact( "OPMODE04_DB".PowerOK.ST00240_RT02_VFD01 )
      I_Contact( "ST00240_2_DB".LT02_VFD01.DRIVE_RUNNING )
   END_RUNG wire#w2
   RUNG wire#powerrail
      Contact( "OPMODE04_DB".PowerOK.ST00240_RT02_VFD01 )
      I_Contact( "ST00240_2_DB".LT02_VFD01.DRIVE_RUNNING )
   END_RUNG wire#w3
   RUNG wire#powerrail
      Contact( "+ST00240.RT02-PX11:4" )
   END_RUNG wire#w4
   RUNG wire#powerrail
      Contact( "+ST00240.RT02-PX12:4" )
   END_RUNG wire#w4
   RUNG wire#powerrail
      Contact( "+ST00240.RT02-PX21:4" )
      Contact( FALSE )
   END_RUNG wire#w5
   RUNG wire#powerrail
      Contact( "+ST00240.CC01-PX21.20:4" )
   END_RUNG wire#w5
   // the same network as SCL:
   "ST00240_RT02_IDB"(PLANT_IDENTIFIER := WSTRING#'+ST00240.RT02',   // "RT_2S2D1P_PD_FB": REMOVED SENSOR "+ST00240.RT02-PX21:4" Use sensor "+ST00240.CC01-PX21.20:4" (Same sensor for CC POS 2)
                      ENABLE_BLOCK := "CONTROL_ON_IDB".CONTROL_ON_DELAYED_1,
                      SAFETY_OK := "IF_SAFE_TO_STND_DB".OPMode04.SafetyOK.ST00240_RT02,
                      HS_FROM_SUCCESSOR := "ST00240_2_DB".HS_FROM_SUCCESSOR,
                      HS_FROM_PREDECESSOR := "ST00240_2_DB".HS_FROM_PREDECESSOR,
                      AUTO_CONVEY_FORWARD := "ST00240_2_DB".LT02.OCCUPIED,
                      ENABLE_FORWARD := "ST00240_2_DB".LT02.POS_UP,
                      ENABLE_REVERSE := "ST00240_2_DB".LT02.POS_UP,
                      ABS_ENABLE_FORWARD := "OPMODE04_DB".PowerOK.ST00240_RT02_VFD01 AND NOT "ST00240_2_DB".LT02_VFD01.DRIVE_RUNNING,
                      ABS_ENABLE_REVERSE := "OPMODE04_DB".PowerOK.ST00240_RT02_VFD01 AND NOT "ST00240_2_DB".LT02_VFD01.DRIVE_RUNNING,
                      PB_FORWARD := #HMI_EXTENSION.Forward,
                      PB_REVERSE := #HMI_EXTENSION.Backward,
                      POS_END_FORWARD_1 := "+ST00240.RT02-PX11:4" OR "+ST00240.RT02-PX12:4",
                      POS_END_REVERSE := ("+ST00240.RT02-PX21:4" AND FALSE) OR "+ST00240.CC01-PX21.20:4",
                      POS_SLOW_FORWARD := "+ST00240.RT02-PX12:4",
                      SELECT_FAST := #HMI_EXTENSION.Fast,
                      "RUN_W/O_ENABLE" := #HMI_EXTENSION.Setup,
                      DRIVE_READY := "ST00240_2_DB".RT02_VFD01.DRIVE_READY,
                      DRIVE_RUNNING := "ST00240_2_DB".RT02_VFD01.DRIVE_RUNNING,
                      EXTERNAL_ALARM := "ST00240_2_DB".Alarm,
                      HIDE_ALARM_MASK := "ST00240_2_DB".RT02_HideAlarmMask,
                      SET_OCC := "ST00240_2_DB".LT02.RT_SET_OCC,
                      RESET_OCC := "ST00240_2_DB".LT02.RT_RESET_OCC,
                      OPMODE_USER_INTERFACE_OUT := "ST00240_2_DB".OPMODE,
                      "GLOBAL_CLOCK&SYSTEM" := "GLOBAL_INFO_IDB".HMI_GLOBAL."Clock&System",
                      IF_HMI := "GLOBAL_RT_2S2D1P_HMI_IF_DB".RT[6],
                      IF_PARA_SET := "ST00240_2_DB".RT02.PARA_SET,
                      HMI_SCREEN_AREA_POINTER := "GLOBAL_HMI_IF_DB".HMI_SCREEN_NO,
                      HMI_SELECT_TIMESTAMP := "GLOBAL_HMI_IF_DB".HMI_SELECT_TIMESTAMP,
                      FORWARD => "ST00240_2_DB".RT02.FORWARD,
                      REVERSE => "ST00240_2_DB".RT02.REVERSE,
                      FAST => "ST00240_2_DB".RT02.FAST,
                      SLOW => "ST00240_2_DB".RT02.SLOW,
                      JOG => "ST00240_2_DB".RT02.JOG,
                      OPEN_BRAKE => "ST00240_2_DB".RT02.OPEN_BRAKE,
                      GENERAL_ALARM => "ST00240_2_DB".RT02.GENERAL_ALARM,
                      HS_TO_SUCCESSOR => "ST00240_2_DB".RT02.HS_TO_SUCCESSOR,
                      HS_TO_PREDECESSOR => "ST00240_2_DB".RT02.HS_TO_PREDECESSOR,
                      DISPLAY_OCCUPIED => "ST00240_2_DB".RT02.DISPLAY_OCCUPIED,
                      DISPLAY_TRANSPORT => "ST00240_2_DB".RT02.DISPLAY_TRANSPORT,
                      DISPLAY_IN_POSITION => "ST00240_2_DB".RT02.DISPLAY_IN_POSITION,
                      DISPLAY_EMPTY => "ST00240_2_DB".RT02.DISPLAY_EMPTY,
                      DISPLAY_OCCCARBODY => "ST00240_2_DB".RT02.DISPLAY_OCCCARBODY,
                      DISPLAY_BLOCKENTRY => "ST00240_2_DB".RT02.DISPLAY_BLOCKENTRY,
                      DISPLAY_BLOCKEXIT => "ST00240_2_DB".RT02.DISPLAY_BLOCKEXIT);
END_REGION

REGION Network 16: RT02 Speed
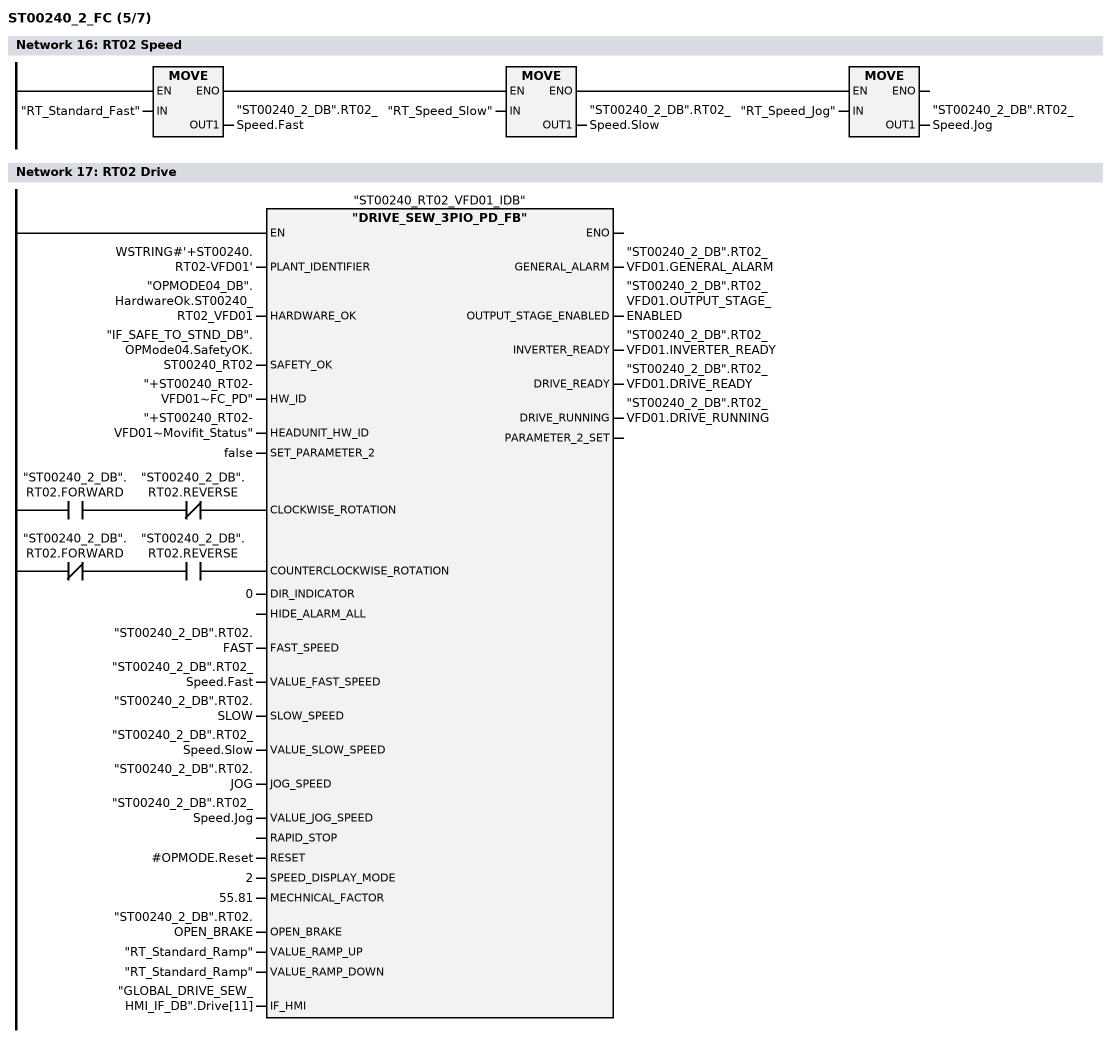
   RUNG wire#powerrail
      Move(in := "RT_Standard_Fast", out1 => "ST00240_2_DB".RT02_Speed.Fast)
      Move(in := "RT_Speed_Slow", out1 => "ST00240_2_DB".RT02_Speed.Slow)
      Move(in := "RT_Speed_Jog", out1 => "ST00240_2_DB".RT02_Speed.Jog)
   END_RUNG
   // the same network as SCL:
   "ST00240_2_DB".RT02_Speed.Fast := "RT_Standard_Fast";
   "ST00240_2_DB".RT02_Speed.Slow := "RT_Speed_Slow";
   "ST00240_2_DB".RT02_Speed.Jog := "RT_Speed_Jog";
END_REGION

REGION Network 17: RT02 Drive
   RUNG wire#powerrail
      "ST00240_RT02_VFD01_IDB"(CLOCKWISE_ROTATION := wire#w1, COUNTERCLOCKWISE_ROTATION := wire#w2, PLANT_IDENTIFIER := WSTRING#'+ST00240.RT02-VFD01', HARDWARE_OK := "OPMODE04_DB".HardwareOk.ST00240_RT02_VFD01, SAFETY_OK := "IF_SAFE_TO_STND_DB".OPMode04.SafetyOK.ST00240_RT02, HW_ID := "+ST00240_RT02-VFD01~FC_PD", HEADUNIT_HW_ID := "+ST00240_RT02-VFD01~Movifit_Status", SET_PARAMETER_2 := false, DIR_INDICATOR := 0, HIDE_ALARM_ALL :=, FAST_SPEED := "ST00240_2_DB".RT02.FAST, VALUE_FAST_SPEED := "ST00240_2_DB".RT02_Speed.Fast, SLOW_SPEED := "ST00240_2_DB".RT02.SLOW, VALUE_SLOW_SPEED := "ST00240_2_DB".RT02_Speed.Slow, JOG_SPEED := "ST00240_2_DB".RT02.JOG, VALUE_JOG_SPEED := "ST00240_2_DB".RT02_Speed.Jog, RAPID_STOP :=, RESET := #OPMODE.Reset, SPEED_DISPLAY_MODE := 2, MECHNICAL_FACTOR := 55.81, OPEN_BRAKE := "ST00240_2_DB".RT02.OPEN_BRAKE, VALUE_RAMP_UP := "RT_Standard_Ramp", VALUE_RAMP_DOWN := "RT_Standard_Ramp", IF_HMI := "GLOBAL_DRIVE_SEW_HMI_IF_DB".Drive[11], GENERAL_ALARM => "ST00240_2_DB".RT02_VFD01.GENERAL_ALARM, OUTPUT_STAGE_ENABLED => "ST00240_2_DB".RT02_VFD01.OUTPUT_STAGE_ENABLED, INVERTER_READY => "ST00240_2_DB".RT02_VFD01.INVERTER_READY, DRIVE_READY => "ST00240_2_DB".RT02_VFD01.DRIVE_READY, DRIVE_RUNNING => "ST00240_2_DB".RT02_VFD01.DRIVE_RUNNING, PARAMETER_2_SET =>)
   END_RUNG
   RUNG wire#powerrail
      Contact( "ST00240_2_DB".RT02.FORWARD )
      I_Contact( "ST00240_2_DB".RT02.REVERSE )
   END_RUNG wire#w1
   RUNG wire#powerrail
      I_Contact( "ST00240_2_DB".RT02.FORWARD )
      Contact( "ST00240_2_DB".RT02.REVERSE )
   END_RUNG wire#w2
   // the same network as SCL:
   "ST00240_RT02_VFD01_IDB"(PLANT_IDENTIFIER := WSTRING#'+ST00240.RT02-VFD01',   // "DRIVE_SEW_3PIO_PD_FB"
                           HARDWARE_OK := "OPMODE04_DB".HardwareOk.ST00240_RT02_VFD01,
                           SAFETY_OK := "IF_SAFE_TO_STND_DB".OPMode04.SafetyOK.ST00240_RT02,
                           HW_ID := "+ST00240_RT02-VFD01~FC_PD",
                           HEADUNIT_HW_ID := "+ST00240_RT02-VFD01~Movifit_Status",
                           SET_PARAMETER_2 := false,
                           CLOCKWISE_ROTATION := "ST00240_2_DB".RT02.FORWARD AND NOT "ST00240_2_DB".RT02.REVERSE,
                           COUNTERCLOCKWISE_ROTATION := NOT "ST00240_2_DB".RT02.FORWARD AND "ST00240_2_DB".RT02.REVERSE,
                           DIR_INDICATOR := 0,
                           FAST_SPEED := "ST00240_2_DB".RT02.FAST,
                           VALUE_FAST_SPEED := "ST00240_2_DB".RT02_Speed.Fast,
                           SLOW_SPEED := "ST00240_2_DB".RT02.SLOW,
                           VALUE_SLOW_SPEED := "ST00240_2_DB".RT02_Speed.Slow,
                           JOG_SPEED := "ST00240_2_DB".RT02.JOG,
                           VALUE_JOG_SPEED := "ST00240_2_DB".RT02_Speed.Jog,
                           RESET := #OPMODE.Reset,
                           SPEED_DISPLAY_MODE := 2,
                           MECHNICAL_FACTOR := 55.81,
                           OPEN_BRAKE := "ST00240_2_DB".RT02.OPEN_BRAKE,
                           VALUE_RAMP_UP := "RT_Standard_Ramp",
                           VALUE_RAMP_DOWN := "RT_Standard_Ramp",
                           IF_HMI := "GLOBAL_DRIVE_SEW_HMI_IF_DB".Drive[11],
                           GENERAL_ALARM => "ST00240_2_DB".RT02_VFD01.GENERAL_ALARM,
                           OUTPUT_STAGE_ENABLED => "ST00240_2_DB".RT02_VFD01.OUTPUT_STAGE_ENABLED,
                           INVERTER_READY => "ST00240_2_DB".RT02_VFD01.INVERTER_READY,
                           DRIVE_READY => "ST00240_2_DB".RT02_VFD01.DRIVE_READY,
                           DRIVE_RUNNING => "ST00240_2_DB".RT02_VFD01.DRIVE_RUNNING);
END_REGION

REGION Network 18: *******************TT02 Control*******************
END_REGION

REGION Network 19: TT02 FB Control
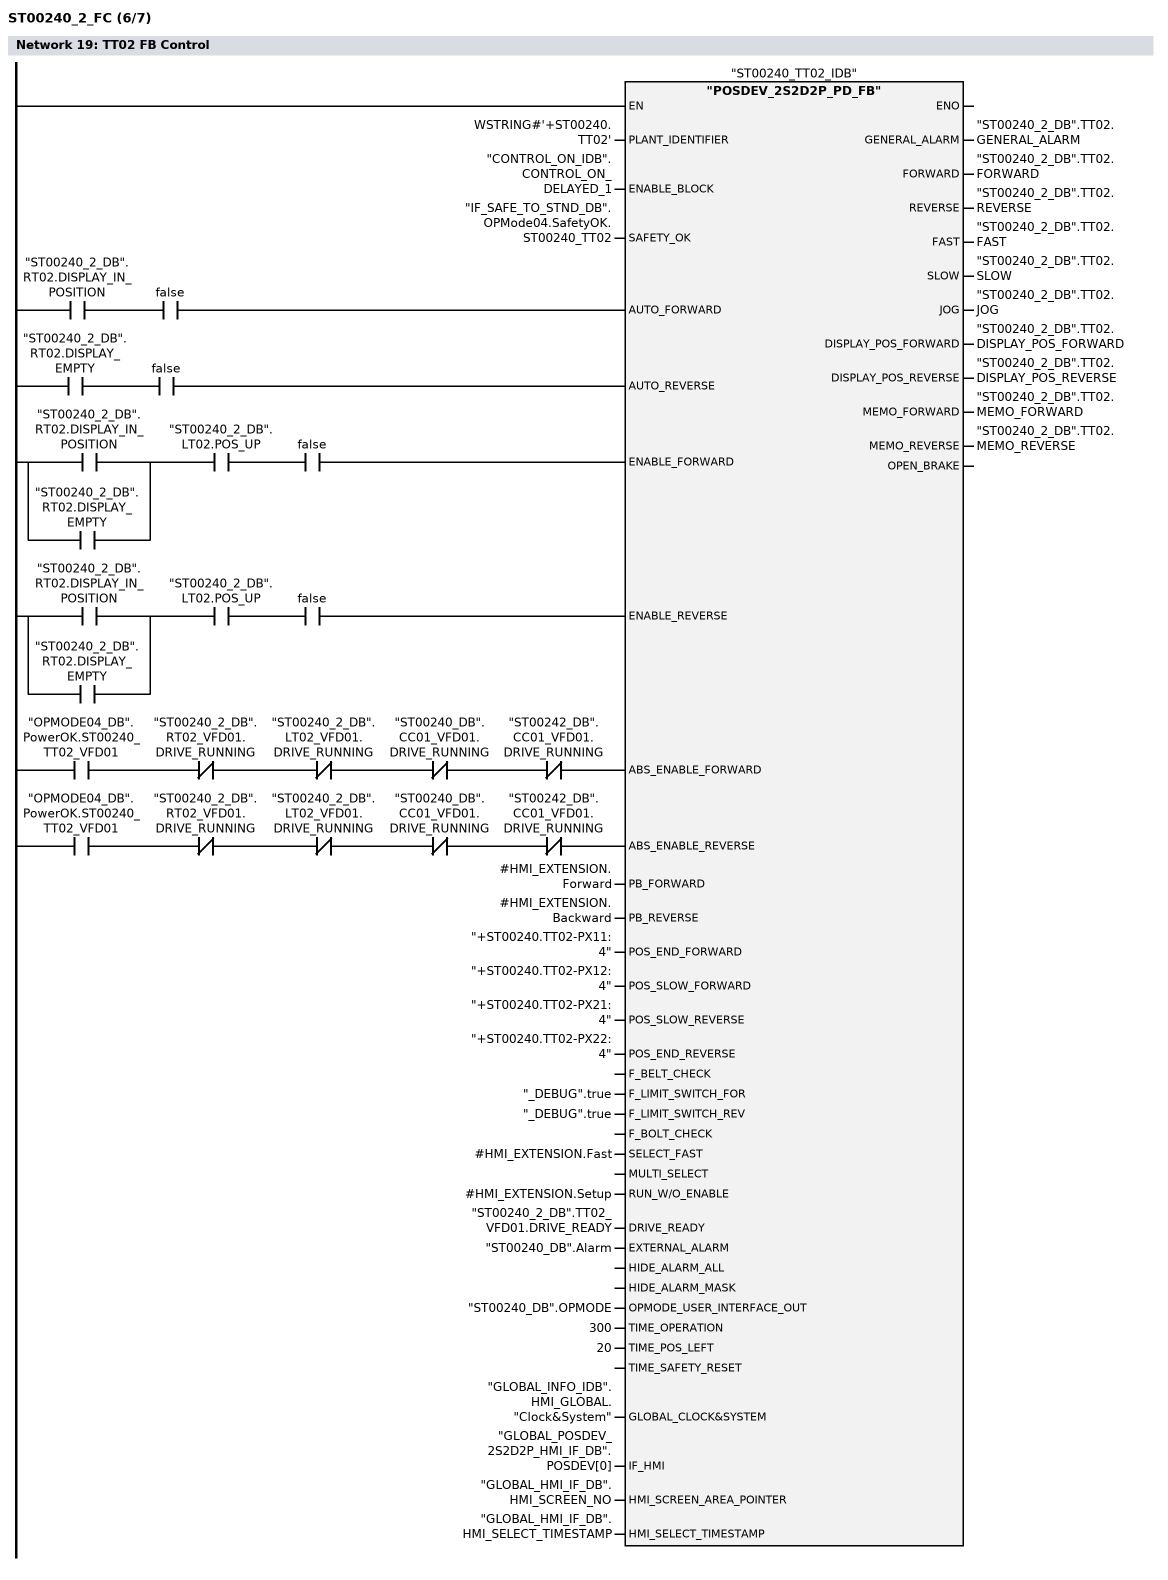
   RUNG wire#powerrail
      "ST00240_TT02_IDB"(AUTO_FORWARD := wire#w1, AUTO_REVERSE := wire#w2, ENABLE_FORWARD := wire#w4, ENABLE_REVERSE := wire#w6, ABS_ENABLE_FORWARD := wire#w7, ABS_ENABLE_REVERSE := wire#w8, PLANT_IDENTIFIER := WSTRING#'+ST00240.TT02', ENABLE_BLOCK := "CONTROL_ON_IDB".CONTROL_ON_DELAYED_1, SAFETY_OK := "IF_SAFE_TO_STND_DB".OPMode04.SafetyOK.ST00240_TT02, PB_FORWARD := #HMI_EXTENSION.Forward, PB_REVERSE := #HMI_EXTENSION.Backward, POS_END_FORWARD := "+ST00240.TT02-PX11:4", POS_SLOW_FORWARD := "+ST00240.TT02-PX12:4", POS_SLOW_REVERSE := "+ST00240.TT02-PX21:4", POS_END_REVERSE := "+ST00240.TT02-PX22:4", F_BELT_CHECK :=, F_LIMIT_SWITCH_FOR := "_DEBUG".true, F_LIMIT_SWITCH_REV := "_DEBUG".true, F_BOLT_CHECK :=, SELECT_FAST := #HMI_EXTENSION.Fast, MULTI_SELECT :=, "RUN_W/O_ENABLE" := #HMI_EXTENSION.Setup, DRIVE_READY := "ST00240_2_DB".TT02_VFD01.DRIVE_READY, EXTERNAL_ALARM := "ST00240_DB".Alarm, HIDE_ALARM_ALL :=, HIDE_ALARM_MASK :=, OPMODE_USER_INTERFACE_OUT := "ST00240_DB".OPMODE, TIME_OPERATION := 300, TIME_POS_LEFT := 20, TIME_SAFETY_RESET :=, "GLOBAL_CLOCK&SYSTEM" := "GLOBAL_INFO_IDB".HMI_GLOBAL."Clock&System", IF_HMI := "GLOBAL_POSDEV_2S2D2P_HMI_IF_DB".POSDEV[0], HMI_SCREEN_AREA_POINTER := "GLOBAL_HMI_IF_DB".HMI_SCREEN_NO, HMI_SELECT_TIMESTAMP := "GLOBAL_HMI_IF_DB".HMI_SELECT_TIMESTAMP, GENERAL_ALARM => "ST00240_2_DB".TT02.GENERAL_ALARM, FORWARD => "ST00240_2_DB".TT02.FORWARD, REVERSE => "ST00240_2_DB".TT02.REVERSE, FAST => "ST00240_2_DB".TT02.FAST, SLOW => "ST00240_2_DB".TT02.SLOW, JOG => "ST00240_2_DB".TT02.JOG, DISPLAY_POS_FORWARD => "ST00240_2_DB".TT02.DISPLAY_POS_FORWARD, DISPLAY_POS_REVERSE => "ST00240_2_DB".TT02.DISPLAY_POS_REVERSE, MEMO_FORWARD => "ST00240_2_DB".TT02.MEMO_FORWARD, MEMO_REVERSE => "ST00240_2_DB".TT02.MEMO_REVERSE, OPEN_BRAKE =>)
   END_RUNG
   RUNG wire#powerrail
      Contact( "ST00240_2_DB".RT02.DISPLAY_IN_POSITION )
      Contact( false )
   END_RUNG wire#w1
   RUNG wire#powerrail
      Contact( "ST00240_2_DB".RT02.DISPLAY_EMPTY )
      Contact( false )
   END_RUNG wire#w2
   RUNG wire#powerrail
      Contact( "ST00240_2_DB".RT02.DISPLAY_IN_POSITION )
      wire#w3
      Contact( "ST00240_2_DB".LT02.POS_UP )
      Contact( false )
   END_RUNG wire#w4
   RUNG wire#powerrail
      Contact( "ST00240_2_DB".RT02.DISPLAY_EMPTY )
   END_RUNG wire#w3
   RUNG wire#powerrail
      Contact( "ST00240_2_DB".RT02.DISPLAY_IN_POSITION )
      wire#w5
      Contact( "ST00240_2_DB".LT02.POS_UP )
      Contact( false )
   END_RUNG wire#w6
   RUNG wire#powerrail
      Contact( "ST00240_2_DB".RT02.DISPLAY_EMPTY )
   END_RUNG wire#w5
   RUNG wire#powerrail
      Contact( "OPMODE04_DB".PowerOK.ST00240_TT02_VFD01 )
      I_Contact( "ST00240_2_DB".RT02_VFD01.DRIVE_RUNNING )
      I_Contact( "ST00240_2_DB".LT02_VFD01.DRIVE_RUNNING )
      I_Contact( "ST00240_DB".CC01_VFD01.DRIVE_RUNNING )
      I_Contact( "ST00242_DB".CC01_VFD01.DRIVE_RUNNING )
   END_RUNG wire#w7
   RUNG wire#powerrail
      Contact( "OPMODE04_DB".PowerOK.ST00240_TT02_VFD01 )
      I_Contact( "ST00240_2_DB".RT02_VFD01.DRIVE_RUNNING )
      I_Contact( "ST00240_2_DB".LT02_VFD01.DRIVE_RUNNING )
      I_Contact( "ST00240_DB".CC01_VFD01.DRIVE_RUNNING )
      I_Contact( "ST00242_DB".CC01_VFD01.DRIVE_RUNNING )
   END_RUNG wire#w8
   // the same network as SCL:
   "ST00240_TT02_IDB"(PLANT_IDENTIFIER := WSTRING#'+ST00240.TT02',   // "POSDEV_2S2D2P_PD_FB"
                      ENABLE_BLOCK := "CONTROL_ON_IDB".CONTROL_ON_DELAYED_1,
                      SAFETY_OK := "IF_SAFE_TO_STND_DB".OPMode04.SafetyOK.ST00240_TT02,
                      AUTO_FORWARD := "ST00240_2_DB".RT02.DISPLAY_IN_POSITION AND false,
                      AUTO_REVERSE := "ST00240_2_DB".RT02.DISPLAY_EMPTY AND false,
                      ENABLE_FORWARD := ("ST00240_2_DB".RT02.DISPLAY_IN_POSITION OR "ST00240_2_DB".RT02.DISPLAY_EMPTY) AND "ST00240_2_DB".LT02.POS_UP AND false,
                      ENABLE_REVERSE := ("ST00240_2_DB".RT02.DISPLAY_IN_POSITION OR "ST00240_2_DB".RT02.DISPLAY_EMPTY) AND "ST00240_2_DB".LT02.POS_UP AND false,
                      ABS_ENABLE_FORWARD := "OPMODE04_DB".PowerOK.ST00240_TT02_VFD01 AND NOT "ST00240_2_DB".RT02_VFD01.DRIVE_RUNNING AND NOT "ST00240_2_DB".LT02_VFD01.DRIVE_RUNNING AND NOT "ST00240_DB".CC01_VFD01.DRIVE_RUNNING AND NOT "ST00242_DB".CC01_VFD01.DRIVE_RUNNING,
                      ABS_ENABLE_REVERSE := "OPMODE04_DB".PowerOK.ST00240_TT02_VFD01 AND NOT "ST00240_2_DB".RT02_VFD01.DRIVE_RUNNING AND NOT "ST00240_2_DB".LT02_VFD01.DRIVE_RUNNING AND NOT "ST00240_DB".CC01_VFD01.DRIVE_RUNNING AND NOT "ST00242_DB".CC01_VFD01.DRIVE_RUNNING,
                      PB_FORWARD := #HMI_EXTENSION.Forward,
                      PB_REVERSE := #HMI_EXTENSION.Backward,
                      POS_END_FORWARD := "+ST00240.TT02-PX11:4",
                      POS_SLOW_FORWARD := "+ST00240.TT02-PX12:4",
                      POS_SLOW_REVERSE := "+ST00240.TT02-PX21:4",
                      POS_END_REVERSE := "+ST00240.TT02-PX22:4",
                      F_LIMIT_SWITCH_FOR := "_DEBUG".true,
                      F_LIMIT_SWITCH_REV := "_DEBUG".true,
                      SELECT_FAST := #HMI_EXTENSION.Fast,
                      "RUN_W/O_ENABLE" := #HMI_EXTENSION.Setup,
                      DRIVE_READY := "ST00240_2_DB".TT02_VFD01.DRIVE_READY,
                      EXTERNAL_ALARM := "ST00240_DB".Alarm,
                      OPMODE_USER_INTERFACE_OUT := "ST00240_DB".OPMODE,
                      TIME_OPERATION := 300,
                      TIME_POS_LEFT := 20,
                      "GLOBAL_CLOCK&SYSTEM" := "GLOBAL_INFO_IDB".HMI_GLOBAL."Clock&System",
                      IF_HMI := "GLOBAL_POSDEV_2S2D2P_HMI_IF_DB".POSDEV[0],
                      HMI_SCREEN_AREA_POINTER := "GLOBAL_HMI_IF_DB".HMI_SCREEN_NO,
                      HMI_SELECT_TIMESTAMP := "GLOBAL_HMI_IF_DB".HMI_SELECT_TIMESTAMP,
                      GENERAL_ALARM => "ST00240_2_DB".TT02.GENERAL_ALARM,
                      FORWARD => "ST00240_2_DB".TT02.FORWARD,
                      REVERSE => "ST00240_2_DB".TT02.REVERSE,
                      FAST => "ST00240_2_DB".TT02.FAST,
                      SLOW => "ST00240_2_DB".TT02.SLOW,
                      JOG => "ST00240_2_DB".TT02.JOG,
                      DISPLAY_POS_FORWARD => "ST00240_2_DB".TT02.DISPLAY_POS_FORWARD,
                      DISPLAY_POS_REVERSE => "ST00240_2_DB".TT02.DISPLAY_POS_REVERSE,
                      MEMO_FORWARD => "ST00240_2_DB".TT02.MEMO_FORWARD,
                      MEMO_REVERSE => "ST00240_2_DB".TT02.MEMO_REVERSE);
END_REGION

REGION Network 20: TT02 Speed
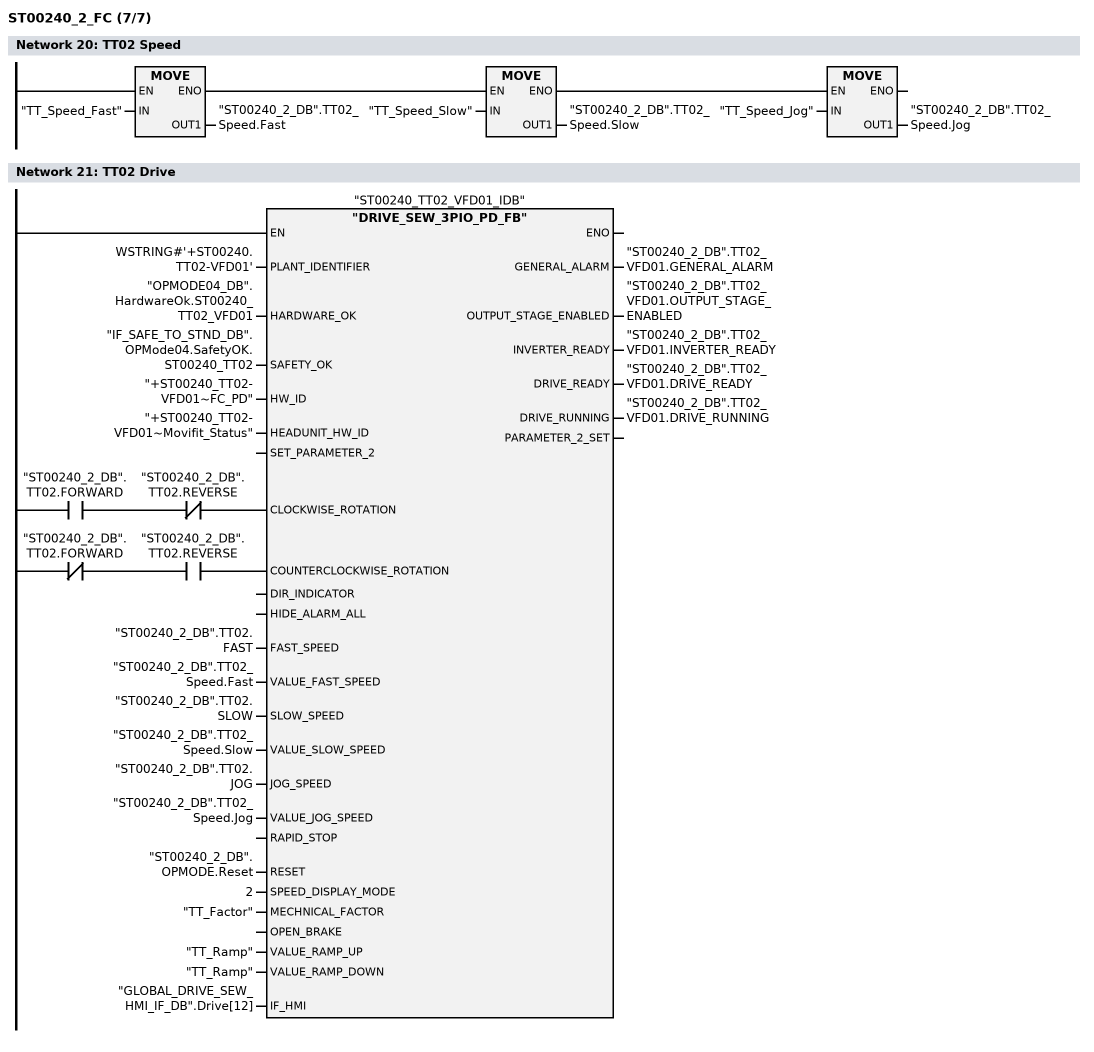
   RUNG wire#powerrail
      Move(in := "TT_Speed_Fast", out1 => "ST00240_2_DB".TT02_Speed.Fast)
      Move(in := "TT_Speed_Slow", out1 => "ST00240_2_DB".TT02_Speed.Slow)
      Move(in := "TT_Speed_Jog", out1 => "ST00240_2_DB".TT02_Speed.Jog)
   END_RUNG
   // the same network as SCL:
   "ST00240_2_DB".TT02_Speed.Fast := "TT_Speed_Fast";
   "ST00240_2_DB".TT02_Speed.Slow := "TT_Speed_Slow";
   "ST00240_2_DB".TT02_Speed.Jog := "TT_Speed_Jog";
END_REGION

REGION Network 21: TT02 Drive
   RUNG wire#powerrail
      "ST00240_TT02_VFD01_IDB"(CLOCKWISE_ROTATION := wire#w1, COUNTERCLOCKWISE_ROTATION := wire#w2, PLANT_IDENTIFIER := WSTRING#'+ST00240.TT02-VFD01', HARDWARE_OK := "OPMODE04_DB".HardwareOk.ST00240_TT02_VFD01, SAFETY_OK := "IF_SAFE_TO_STND_DB".OPMode04.SafetyOK.ST00240_TT02, HW_ID := "+ST00240_TT02-VFD01~FC_PD", HEADUNIT_HW_ID := "+ST00240_TT02-VFD01~Movifit_Status", SET_PARAMETER_2 :=, DIR_INDICATOR :=, HIDE_ALARM_ALL :=, FAST_SPEED := "ST00240_2_DB".TT02.FAST, VALUE_FAST_SPEED := "ST00240_2_DB".TT02_Speed.Fast, SLOW_SPEED := "ST00240_2_DB".TT02.SLOW, VALUE_SLOW_SPEED := "ST00240_2_DB".TT02_Speed.Slow, JOG_SPEED := "ST00240_2_DB".TT02.JOG, VALUE_JOG_SPEED := "ST00240_2_DB".TT02_Speed.Jog, RAPID_STOP :=, RESET := "ST00240_2_DB".OPMODE.Reset, SPEED_DISPLAY_MODE := 2, MECHNICAL_FACTOR := "TT_Factor", OPEN_BRAKE :=, VALUE_RAMP_UP := "TT_Ramp", VALUE_RAMP_DOWN := "TT_Ramp", IF_HMI := "GLOBAL_DRIVE_SEW_HMI_IF_DB".Drive[12], GENERAL_ALARM => "ST00240_2_DB".TT02_VFD01.GENERAL_ALARM, OUTPUT_STAGE_ENABLED => "ST00240_2_DB".TT02_VFD01.OUTPUT_STAGE_ENABLED, INVERTER_READY => "ST00240_2_DB".TT02_VFD01.INVERTER_READY, DRIVE_READY => "ST00240_2_DB".TT02_VFD01.DRIVE_READY, DRIVE_RUNNING => "ST00240_2_DB".TT02_VFD01.DRIVE_RUNNING, PARAMETER_2_SET =>)
   END_RUNG
   RUNG wire#powerrail
      Contact( "ST00240_2_DB".TT02.FORWARD )
      I_Contact( "ST00240_2_DB".TT02.REVERSE )
   END_RUNG wire#w1
   RUNG wire#powerrail
      I_Contact( "ST00240_2_DB".TT02.FORWARD )
      Contact( "ST00240_2_DB".TT02.REVERSE )
   END_RUNG wire#w2
   // the same network as SCL:
   "ST00240_TT02_VFD01_IDB"(PLANT_IDENTIFIER := WSTRING#'+ST00240.TT02-VFD01',   // "DRIVE_SEW_3PIO_PD_FB"
                           HARDWARE_OK := "OPMODE04_DB".HardwareOk.ST00240_TT02_VFD01,
                           SAFETY_OK := "IF_SAFE_TO_STND_DB".OPMode04.SafetyOK.ST00240_TT02,
                           HW_ID := "+ST00240_TT02-VFD01~FC_PD",
                           HEADUNIT_HW_ID := "+ST00240_TT02-VFD01~Movifit_Status",
                           CLOCKWISE_ROTATION := "ST00240_2_DB".TT02.FORWARD AND NOT "ST00240_2_DB".TT02.REVERSE,
                           COUNTERCLOCKWISE_ROTATION := NOT "ST00240_2_DB".TT02.FORWARD AND "ST00240_2_DB".TT02.REVERSE,
                           FAST_SPEED := "ST00240_2_DB".TT02.FAST,
                           VALUE_FAST_SPEED := "ST00240_2_DB".TT02_Speed.Fast,
                           SLOW_SPEED := "ST00240_2_DB".TT02.SLOW,
                           VALUE_SLOW_SPEED := "ST00240_2_DB".TT02_Speed.Slow,
                           JOG_SPEED := "ST00240_2_DB".TT02.JOG,
                           VALUE_JOG_SPEED := "ST00240_2_DB".TT02_Speed.Jog,
                           RESET := "ST00240_2_DB".OPMODE.Reset,
                           SPEED_DISPLAY_MODE := 2,
                           MECHNICAL_FACTOR := "TT_Factor",
                           VALUE_RAMP_UP := "TT_Ramp",
                           VALUE_RAMP_DOWN := "TT_Ramp",
                           IF_HMI := "GLOBAL_DRIVE_SEW_HMI_IF_DB".Drive[12],
                           GENERAL_ALARM => "ST00240_2_DB".TT02_VFD01.GENERAL_ALARM,
                           OUTPUT_STAGE_ENABLED => "ST00240_2_DB".TT02_VFD01.OUTPUT_STAGE_ENABLED,
                           INVERTER_READY => "ST00240_2_DB".TT02_VFD01.INVERTER_READY,
                           DRIVE_READY => "ST00240_2_DB".TT02_VFD01.DRIVE_READY,
                           DRIVE_RUNNING => "ST00240_2_DB".TT02_VFD01.DRIVE_RUNNING);
END_REGION
END_FUNCTION
